(* CODESYS project ElevatorProblem.project

Project tree, tasks and I/O mapping:
  Device : Elmo Platinum Maestro, Elmo Motion Control, version 1.0.0.2
    application Application
      libraries: Standard, * (System)
      task MainTask (cyclic, interval t#100ms, priority 1) calls PLC_PRG, PLC_PRG
      task VISU_TASK (cyclic, interval 100 ms, priority 31) calls VisuElems.Visu_Prg
      program PLC_PRG [ST]
      01_Enumerator/
        data type eFloor
        data type eMOVESTOP
        data type eElevatorType
        data type eButton
        data type eUPDOWN
      02_Structure/
        data type stElevator
        data type stFloor
        data type stFloorRequest
      03_Module/
        function block FB_Elevator [ST]: M_ColorElevator, pCurrentFloor, M_Move, M_ButtonClicked, pColorButtons, pDestinPos, pB1Invisible, M_ShowClickedButton, M_FloorReached, M_DetermineNextFloor, pCurrentRequest, pMoving, pDirection, pCurrentDestin, pRequest, pCurrentPos, pCurrentPeople, pMaxPeople
        function block FB_ElevatorGuests [ST]: pColorButtons, pB1Invisible, pMaxPeople
        function block FB_Floor [ST]: pTopInvisible, pBottomInvisible, pFloorNumber, pPeople
        function block FB_FloorTop [ST]: pTopInvisible
        function block FB_FloorBottom [ST]: pBottomInvisible
        function block FB_Building [ST]: M_RequestExecuted, pFloorRequestedQueue, M_NewFloorRequest, M_AssignElevators, M_Distance
      visualisation Visualization
      visualisation Elevator
      visualisation Floor
    Elmo_Master_Device : Elmo Master Device, Elmo, version 1.0.0.2
  libraries: VisuSymbols, 3.5.10.0 (System)
  text list GlobalTextList
*)

// Device/Application/01_Enumerator/eFloor
TYPE eFloor :
(
	Wait := -1,
	B1 := 0,
	F1 := 1,
	F2 := 2,
	F3 := 3,
	F4 := 4,
	F5 := 5
);
END_TYPE

// Device/Application/01_Enumerator/eMOVESTOP
TYPE eMOVESTOP :
(
	WAITING := 0, // doors are open -> people can get on and off
	MOVING := 1,
	STOPPING := 2
);
END_TYPE

// Device/Application/02_Structure/stElevator
TYPE stElevator :
STRUCT
	uiElevatorType : UINT;
	dwColorElevator : DWORD;
	dwColorButtons : DWORD;
	uiCurrentPos : UINT := 0;
	iDestinPos : UINT := 0;
	uiCurrentPeople : UINT;
	uiCurrentFloor : eFloor;
	xMoving : BOOL;
	xB1Access : BOOL;
	
	// Bools and trigger for buttons
	trig_ButtonF1 : R_Trig;
	xF1 : BOOL;
	xF1Clicked : BOOL;
	trig_ButtonF2 : R_Trig;
	xF2 : BOOL;
	xF2Clicked : BOOL;
	trig_ButtonF3 : R_Trig;
	xF3 : BOOL;
	xF3Clicked : BOOL;
	trig_ButtonF4 : R_Trig;
	xF4 : BOOL;
	xF4Clicked : BOOL;
	trig_ButtonF5 : R_Trig;
	xF5 : BOOL;
	xF5Clicked : BOOL;
	trig_ButtonB1 : R_Trig;
	xB1 : BOOL;
	xB1Clicked : BOOL;
	trig_ButtonClose : R_Trig;
	xClose : BOOL;
	trig_ButtonOpen : R_Trig;
	xOpen : BOOL;
		
END_STRUCT
END_TYPE

// Device/Application/01_Enumerator/eElevatorType
{attribute 'qualified_only'}
{attribute 'strict'}
TYPE eElevatorType :
(
	GUEST := 1,
	FREIGHT := 0
);
END_TYPE

// Device/Application/02_Structure/stFloor
TYPE stFloor :
STRUCT
	uiFloorNumber : UINT;
	uiPeople : UINT;
	
	xTopInvisible : BOOL;
	xBottomInvisible : BOOL;
	
	trig_ButtonUP : R_Trig;
	xUP : BOOL;
	xUpClicked : BOOL;
	trig_ButtonDOWN : R_Trig;
	xDOWN : BOOL;
	xDownClicked : BOOL;
	
	trig_ButtonPeople : R_Trig;
	xPeople : BOOL;
	trig_ButtonPeopleMinus : R_Trig;
	xPeopleMinus : BOOL;
	
END_STRUCT
END_TYPE

// Device/Application/01_Enumerator/eButton
{attribute 'qualified_only'}
{attribute 'strict'}
TYPE eButton :
(
	B1 := 0,
	F1 := 1,
	F2 := 2,
	F3 := 3,
	F4 := 4,
	F5 := 5,
	CLOSE := 6,
	OPEN := 7
);
END_TYPE

// Device/Application/01_Enumerator/eUPDOWN
{attribute 'qualified_only'}
{attribute 'strict'}
TYPE eUPDOWN :
(
	Wait := -1,
	UP := 0,
	DOWN := 1
);
END_TYPE

// Device/Application/02_Structure/stFloorRequest
TYPE stFloorRequest :
STRUCT
	eFloor : eFloor := -1;
    eUPDOWN : eUPDOWN := -1;
END_STRUCT
END_TYPE

// Device/Application/PLC_PRG
PROGRAM PLC_PRG
VAR
	(* Object declarations *)
	fbElevatorGuests : ARRAY [1..uiObject] OF FB_ElevatorGuests; // Elevator 1 and 2
	stElevatorGuestsData : ARRAY [1..uiObject] OF stElevator;	// Data for elevator 1 and 2
	
	fbElevator : FB_Elevator;	// Elevator 3
	stElevatorData : stElevator;	// Data for Elevator 3
	
	fbBuilding : FB_Building;	// Building
	fbAllElevators : ARRAY [1..3] OF FB_Elevator;	// Array with all Elevators of Building
	fbAllFloors : ARRAY[0..5] OF FB_Floor;
	
	fbFloor : ARRAY [1..uiObjectFloor] OF FB_Floor;	// Floors 1 to 4
	stFloorData : ARRAY [1..uiObjectFloor] OF stFLoor;	// Data for Floor 1 to 4
	
	fbFloorTop : FB_FloorTop;	// Floor 5
	stFloorTopData : stFloor;	// Data for Floor 5
	
	fbFloorBottom : FB_FloorBottom;	// Floor B1 aka 0
	stFloorBottomData : stFloor;	// Data for Floor B1
	
	(* Variables for handling elevator movements and requests *)
	xButtonsClicked : ARRAY[0..5] OF BOOL;	// Array for clicked buttons
	CommandToElevator : ARRAY [1..3] OF stFloorRequest;	// Array for Floor Requests to Elevator
	
	// new Floor Requests
	stNewFloorRequest : stFloorRequest;
	eRequestedFloor : stFloorRequest;
	xFloorRequestClicked : ARRAY[1..10] OF BOOL;
	
	// helper variables
	iCnt : UINT;	// counter Variable
	uiPeopleElevators : ARRAY[1..3] OF UINT;
	uiPeopleFloors : ARRAY[0..5] OF UINT;
	

	
END_VAR
VAR CONSTANT
	uiObject : UINT := 2;
	uiObjectFloor : UINT :=4;
END_VAR

// FLOORS
FOR iCnt := 1 TO uiObjectFloor BY 1 DO
	fbFloor[iCnt].pFloorNumber := iCnt;
	stFloorData[iCnt].uiPeople := fbFloor[iCnt].pPeople;
	stFloorData[iCnt].uiFloorNumber := fbFloor[iCnt].pFloorNumber;
	stFloorData[iCnt].xBottomInvisible := fbFloor[iCnt].pBottomInvisible;
	stFloorData[iCnt].xTopInvisible := fbFloor[iCnt].pTopInvisible;
	stFloorData[iCnt].trig_ButtonDOWN(CLK := stFloorData[iCnt].xDOWN);
	stFloorData[iCnt].trig_ButtonUP(CLK := stFloorData[iCnt].xUP);
	stFloorData[iCnt].trig_ButtonPeople(CLK := stFloorData[iCnt].xPeople);
	stFloorData[iCnt].trig_ButtonPeopleMinus(CLK := stFloorData[iCnt].xPeopleMinus);
	IF stFloorData[iCnt].trig_ButtonDOWN.Q THEN
		stNewFloorRequest.eFloor := fbFloor[iCnt].pFloorNumber;
		stNewFloorRequest.eUPDOWN := eUPDOWN.DOWN;
		fbBuilding.M_NewFloorRequest(stNewFloorRequest);
		xFloorRequestClicked[iCnt*2] := TRUE;
	ELSIF stFloorData[iCnt].trig_ButtonUP.Q THEN
		stNewFloorRequest.eFloor := fbFloor[iCnt].pFloorNumber;
		stNewFloorRequest.eUPDOWN := eUPDOWN.UP;
		fbBuilding.M_NewFloorRequest(stNewFloorRequest);
		xFloorRequestClicked[(iCnt*2)+1] := TRUE;
	END_IF
	IF stFloorData[iCnt].trig_ButtonPeople.Q THEN
		fbFloor[iCnt].pPeople := fbFloor[iCnt].pPeople + 1;
	END_IF
	IF stFloorData[iCnt].trig_ButtonPeopleMinus.Q THEN
		IF fbFloor[iCnt].pPeople > 0 THEN
			fbFloor[iCnt].pPeople := fbFloor[iCnt].pPeople - 1;
		END_IF
	END_IF
	stFloorData[iCnt].xDownClicked := xFloorRequestClicked[iCnt*2];
	stFloorData[iCnt].xUpClicked := xFloorRequestClicked[(iCnt*2)+1];
	
	
END_FOR
// Top Floor
fbFloorTop.pFloorNumber := 5;
stFloorTopData.uiPeople := fbFloorTop.pPeople;
stFloorTopData.uiFloorNumber := fbFloorTop.pFloorNumber;
stFloorTopData.xBottomInvisible := fbFloorTop.pBottomInvisible;
stFloorTopData.xTopInvisible := fbFloorTop.pTopInvisible;
stFloorTopData.trig_ButtonDOWN(CLK := stFloorTopData.xDOWN);
stFloorTopData.trig_ButtonPeople(CLK := stFloorTopData.xPeople);
stFloorTopData.trig_ButtonPeopleMinus(CLK := stFloorTopData.xPeopleMinus);
IF stFloorTopData.trig_ButtonDOWN.Q THEN
	stNewFloorRequest.eFloor := fbFloorTop.pFloorNumber;
	stNewFloorRequest.eUPDOWN := eUPDOWN.DOWN;
	fbBuilding.M_NewFloorRequest(stNewFloorRequest);
	xFloorRequestClicked[10] := TRUE;
END_IF
IF stFloorTopData.trig_ButtonPeople.Q THEN
	fbFloorTop.pPeople := fbFloorTop.pPeople + 1;
END_IF
IF stFloorTopData.trig_ButtonPeopleMinus.Q THEN
	IF fbFloorTop.pPeople > 0 THEN
		fbFloorTop.pPeople := fbFloorTop.pPeople - 1;
	END_IF
END_IF
stFloorTopData.xDownClicked := xFloorRequestClicked[10];
// Bottom Floor
fbFloorBottom.pFloorNumber := 0;
stFloorBottomData.uiPeople := fbFloorBottom.pPeople;
stFloorBottomData.uiFloorNumber := fbFloorBottom.pFloorNumber;
stFloorBottomData.xBottomInvisible := fbFloorBottom.pBottomInvisible;
stFloorBottomData.xTopInvisible := fbFloorBottom.pTopInvisible;
stFloorBottomData.trig_ButtonUP(CLK := stFloorBottomData.xUP);
stFloorBottomData.trig_ButtonPeople(CLK := stFloorBottomData.xPeople);
stFloorBottomData.trig_ButtonPeopleMinus(CLK := stFloorBottomData.xPeopleMinus);
IF stFloorBottomData.trig_ButtonUP.Q THEN
	stNewFloorRequest.eFloor := fbFloorBottom.pFloorNumber;
	stNewFloorRequest.eUPDOWN := eUPDOWN.UP;
	fbBuilding.M_NewFloorRequest(stNewFloorRequest);
	xFloorRequestClicked[1] := TRUE;
END_IF
IF stFloorBottomData.trig_ButtonPeople.Q THEN
	fbFloorBottom.pPeople := fbFloorBottom.pPeople + 1;
END_IF
IF stFloorBottomData.trig_ButtonPeopleMinus.Q THEN
	IF fbFloorBottom.pPeople > 0 THEN
		fbFloorBottom.pPeople := fbFloorBottom.pPeople - 1;
	END_IF
END_IF
stFloorBottomData.xUpClicked := xFloorRequestClicked[1];



// Building
fbAllFloors[0] := fbFloorBottom;
fbAllFloors[1] := fbFloor[1];
fbAllFloors[2] := fbFloor[2];
fbAllFloors[3] := fbFloor[3];
fbAllFloors[4] := fbFloor[4];
fbAllFloors[5] := fbFloorTop;
fbBuilding.fbFloors := fbAllFloors;
fbAllElevators[1] := fbElevatorGuests[1];
fbAllElevators[2] := fbElevatorGuests[2];
fbAllElevators[3] := fbElevator;
fbBuilding.fbElevators := fbAllElevators;
CommandToElevator := fbBuilding.M_AssignElevators();

// ELEVATORS
// guest elevators
FOR iCnt := 1 TO uiObject BY 1 DO
	// Floor Request
	fbElevatorGuests[iCnt].pCurrentRequest := CommandToElevator[iCnt];
	IF CommandToElevator[iCnt].eFloor <> -1 THEN
		fbElevatorGuests[iCnt].pRequest := TRUE;
		fbElevatorGuests[iCnt].M_DetermineNextFloor();
		fbAllElevators[1] := fbElevatorGuests[1];
		fbAllElevators[2] := fbElevatorGuests[2];
		fbBuilding.fbElevators := fbAllElevators;
	ELSE
		fbElevatorGuests[iCnt].pRequest := FALSE;
	END_IF

	// transfer of general data from the object to the visualization struct
	stElevatorGuestsData[iCnt].xB1Access := fbElevatorGuests[iCnt].pB1Invisible;
	stElevatorGuestsData[iCnt].uiCurrentFloor := fbElevatorGuests[iCnt].pCurrentFloor;
	stElevatorGuestsData[iCnt].dwColorElevator := fbElevatorGuests[iCnt].M_ColorElevator();
	stElevatorGuestsData[iCnt].dwColorButtons := fbElevatorGuests[iCnt].pColorButtons;
	stElevatorGuestsData[iCnt].uiCurrentPeople := fbElevatorGuests[iCnt].pCurrentPeople;
	// MOVE
	stElevatorGuestsData[iCnt].uiCurrentPos := fbElevatorGuests[iCnt].M_Move();

	// Buttons configuration
	stElevatorGuestsData[iCnt].xMoving := fbElevatorGuests[iCnt].xMoving;
	stElevatorGuestsData[iCnt].trig_ButtonF1(CLK := stElevatorGuestsData[iCnt].xF1);
	stElevatorGuestsData[iCnt].trig_ButtonF2(CLK := stElevatorGuestsData[iCnt].xF2);
	stElevatorGuestsData[iCnt].trig_ButtonF3(CLK := stElevatorGuestsData[iCnt].xF3);
	stElevatorGuestsData[iCnt].trig_ButtonF4(CLK := stElevatorGuestsData[iCnt].xF4);
	stElevatorGuestsData[iCnt].trig_ButtonF5(CLK := stElevatorGuestsData[iCnt].xF5);
	stElevatorGuestsData[iCnt].trig_ButtonB1(CLK := stElevatorGuestsData[iCnt].xB1);
	stElevatorGuestsData[iCnt].trig_ButtonClose(CLK := stElevatorGuestsData[iCnt].xClose);
	stElevatorGuestsData[iCnt].trig_ButtonOpen(CLK := stElevatorGuestsData[iCnt].xOpen);
	IF stElevatorGuestsData[iCnt].trig_ButtonF1.Q THEN
		fbElevatorGuests[iCnt].iiPressedButton := eButton.F1;
		fbElevatorGuests[iCnt].M_ButtonClicked(fbElevatorGuests[iCnt].iiPressedButton);
	ELSIF stElevatorGuestsData[iCnt].trig_ButtonF2.Q THEN
		fbElevatorGuests[iCnt].iiPressedButton := eButton.F2;
		fbElevatorGuests[iCnt].M_ButtonClicked(fbElevatorGuests[iCnt].iiPressedButton);
	ELSIF stElevatorGuestsData[iCnt].trig_ButtonF3.Q THEN
		fbElevatorGuests[iCnt].iiPressedButton := eButton.F3;
		fbElevatorGuests[iCnt].M_ButtonClicked(fbElevatorGuests[iCnt].iiPressedButton);
	ELSIF stElevatorGuestsData[iCnt].trig_ButtonF4.Q THEN
		fbElevatorGuests[iCnt].iiPressedButton := eButton.F4;
		fbElevatorGuests[iCnt].M_ButtonClicked(fbElevatorGuests[iCnt].iiPressedButton);
	ELSIF stElevatorGuestsData[iCnt].trig_ButtonF5.Q THEN
		fbElevatorGuests[iCnt].iiPressedButton := eButton.F5;
		fbElevatorGuests[iCnt].M_ButtonClicked(fbElevatorGuests[iCnt].iiPressedButton);
	ELSIF stElevatorGuestsData[iCnt].trig_ButtonB1.Q THEN
		fbElevatorGuests[iCnt].iiPressedButton := eButton.B1;
		fbElevatorGuests[iCnt].M_ButtonClicked(fbElevatorGuests[iCnt].iiPressedButton);
	ELSIF stElevatorGuestsData[iCnt].trig_ButtonClose.Q THEN
		fbElevatorGuests[iCnt].iiPressedButton := eButton.CLOSE;
		fbElevatorGuests[iCnt].M_ButtonClicked(fbElevatorGuests[iCnt].iiPressedButton);
	ELSIF stElevatorGuestsData[iCnt].trig_ButtonOpen.Q THEN
		fbElevatorGuests[iCnt].iiPressedButton := eButton.OPEN;
		fbElevatorGuests[iCnt].M_ButtonClicked(fbElevatorGuests[iCnt].iiPressedButton);
	ELSE
		fbElevatorGuests[iCnt].iiPressedButton := -1;
	END_IF
	
	// Remove request if executed ( if the current status of Requested is False, but before Move() it was true)
	IF NOT fbElevatorGuests[iCnt].pRequest AND fbAllElevators[iCnt].pRequest THEN
		eRequestedFloor := fbElevatorGuests[iCnt].pCurrentRequest;
		IF fbElevatorGuests[iCnt].pCurrentFloor = eRequestedFloor.eFloor THEN
			fbBuilding.M_RequestExecuted(eRequestedFloor);
			// update people on all floors and elevators
			
			uiPeopleElevators := fbBuilding.PeopleToElevator;
			fbElevatorGuests[1].pCurrentPeople := uiPeopleElevators[1];
			fbElevatorGuests[2].pCurrentPeople := uiPeopleElevators[2];
			fbElevator.pCurrentPeople := uiPeopleElevators[3];
			uiPeopleFloors := fbBuilding.PeopleToFloor;
			fbFloorBottom.pPeople := uiPeopleFloors[0];
			fbFloor[1].pPeople := uiPeopleFloors[1];
			fbFloor[2].pPeople := uiPeopleFloors[2];
			fbFloor[3].pPeople := uiPeopleFloors[3];
			fbFloor[4].pPeople := uiPeopleFloors[4];
			fbFloorTop.pPeople := uiPeopleFloors[5];
			
		END_IF
		// untoggle Floor button (F1-F4)
		IF eRequestedFloor.eFloor > eFloor.B1 AND eRequestedFloor.eFloor < eFloor.F5 THEN
			IF eRequestedFloor.eUPDOWN = eUPDOWN.DOWN THEN
				stFloorData[eRequestedFloor.eFloor].xDOWN := FALSE;
				xFloorRequestClicked[eRequestedFloor.eFloor*2] := FALSE;
			ELSIF eRequestedFloor.eUPDOWN = eUPDOWN.UP THEN
				stFloorData[eRequestedFloor.eFloor].xUP := FALSE;
				xFloorRequestClicked[eRequestedFloor.eFloor*2+1] := FALSE;
			END_IF
			// shouldn't happen because not reachable for guest elevators
		ELSIF eRequestedFloor.eFloor = eFloor.B1 THEN
			stFloorBottomData.xUP := FALSE;
			xFloorRequestClicked[1] := FALSE;
		ELSIF eRequestedFloor.eFloor = eFloor.F5 THEN
			stFloorTopData.xDOWN := FALSE;
			xFloorRequestClicked[10] := FALSE;
		END_IF		
	END_IF
	
	// Button style
	xButtonsClicked := fbElevatorGuests[iCnt].M_ShowClickedButton();
	stElevatorGuestsData[iCnt].xB1Clicked := xButtonsClicked[0];
	stElevatorGuestsData[iCnt].xF1Clicked := xButtonsClicked[1];
	stElevatorGuestsData[iCnt].xF2Clicked := xButtonsClicked[2];
	stElevatorGuestsData[iCnt].xF3Clicked := xButtonsClicked[3];
	stElevatorGuestsData[iCnt].xF4Clicked := xButtonsClicked[4];
	stElevatorGuestsData[iCnt].xF5Clicked := xButtonsClicked[5];
	
END_FOR

//  Freight Elevator 
// Floor request
IF CommandToElevator[3].eFloor <> -1 THEN
	fbElevator.pCurrentRequest := CommandToElevator[3];
	fbElevator.pRequest := TRUE;
	fbElevator.M_DetermineNextFloor();
	fbAllElevators[3] := fbElevator;
	fbBuilding.fbElevators := fbAllElevators;
END_IF
// general properites
stElevatorData.xB1Access := fbElevator.pB1Invisible;
stElevatorData.uiCurrentFloor := fbElevator.pCurrentFloor;
stElevatorData.dwColorElevator := fbElevator.M_ColorElevator();
stElevatorData.dwColorButtons := fbElevator.pColorButtons;
stElevatorData.uiCurrentPeople := fbElevator.pCurrentPeople;
// MOVE
stElevatorData.uiCurrentPos := fbElevator.M_Move();
// Button linking
stElevatorData.xMoving := fbElevator.xMoving;
stElevatorData.trig_ButtonF1(CLK := stElevatorData.xF1);
stElevatorData.trig_ButtonF2(CLK := stElevatorData.xF2);
stElevatorData.trig_ButtonF3(CLK := stElevatorData.xF3);
stElevatorData.trig_ButtonF4(CLK := stElevatorData.xF4);
stElevatorData.trig_ButtonF5(CLK := stElevatorData.xF5);
stElevatorData.trig_ButtonB1(CLK := stElevatorData.xB1);
stElevatorData.trig_ButtonClose(CLK := stElevatorData.xClose);
stElevatorData.trig_ButtonOpen(CLK := stElevatorData.xOpen);
IF stElevatorData.trig_ButtonF1.Q THEN
	fbElevator.iiPressedButton := eButton.F1;
	fbElevator.M_ButtonClicked(fbElevator.iiPressedButton);
ELSIF stElevatorData.trig_ButtonF2.Q THEN
	fbElevator.iiPressedButton := eButton.F2;
	fbElevator.M_ButtonClicked(fbElevator.iiPressedButton);
ELSIF stElevatorData.trig_ButtonF3.Q THEN
	fbElevator.iiPressedButton := eButton.F3;
	fbElevator.M_ButtonClicked(fbElevator.iiPressedButton);
ELSIF stElevatorData.trig_ButtonF4.Q THEN
	fbElevator.iiPressedButton := eButton.F4;
	fbElevator.M_ButtonClicked(fbElevator.iiPressedButton);
ELSIF stElevatorData.trig_ButtonF5.Q THEN
	fbElevator.iiPressedButton := eButton.F5;
	fbElevator.M_ButtonClicked(fbElevator.iiPressedButton);
ELSIF stElevatorData.trig_ButtonB1.Q THEN
	fbElevator.iiPressedButton := eButton.B1;
	fbElevator.M_ButtonClicked(fbElevator.iiPressedButton);
ELSIF stElevatorData.trig_ButtonClose.Q THEN
	fbElevator.iiPressedButton := eButton.CLOSE;
	fbElevator.M_ButtonClicked(fbElevator.iiPressedButton);
ELSIF stElevatorData.trig_ButtonOpen.Q THEN
	fbElevator.iiPressedButton := eButton.OPEN;
	fbElevator.M_ButtonClicked(fbElevator.iiPressedButton);
ELSE
	fbElevator.iiPressedButton := -1;
END_IF
// button style depending on clicked or not
xButtonsClicked := fbElevator.M_ShowClickedButton();
stElevatorData.xB1Clicked := xButtonsClicked[0];
stElevatorData.xF1Clicked := xButtonsClicked[1];
stElevatorData.xF2Clicked := xButtonsClicked[2];
stElevatorData.xF3Clicked := xButtonsClicked[3];
stElevatorData.xF4Clicked := xButtonsClicked[4];
stElevatorData.xF5Clicked := xButtonsClicked[5];

// Remove request if executed
IF NOT fbElevator.pRequest AND fbAllElevators[3].pRequest THEN
	eRequestedFloor := fbElevator.pCurrentRequest;
	IF fbElevator.pCurrentFloor = eRequestedFloor.eFloor THEN
		fbBuilding.M_RequestExecuted(eRequestedFloor);// update people on all floors and elevators
		uiPeopleElevators := fbBuilding.PeopleToElevator;
		fbElevatorGuests[1].pCurrentPeople := uiPeopleElevators[1];
		fbElevatorGuests[2].pCurrentPeople := uiPeopleElevators[2];
		fbElevator.pCurrentPeople := uiPeopleElevators[3];
		uiPeopleFloors := fbBuilding.PeopleToFloor;
		fbFloorBottom.pPeople := uiPeopleFloors[0];
		fbFloor[1].pPeople := uiPeopleFloors[1];
		fbFloor[2].pPeople := uiPeopleFloors[2];
		fbFloor[3].pPeople := uiPeopleFloors[3];
		fbFloor[4].pPeople := uiPeopleFloors[4];
		fbFloorTop.pPeople := uiPeopleFloors[5];
	END_IF
	// untoggle Floor button (F1-F4)
	IF eRequestedFloor.eFloor > eFloor.B1 AND eRequestedFloor.eFloor < eFloor.F5 THEN
		IF eRequestedFloor.eUPDOWN = eUPDOWN.DOWN THEN
			stFloorData[eRequestedFloor.eFloor].xDOWN := FALSE;
			xFloorRequestClicked[eRequestedFloor.eFloor*2] := FALSE;
		ELSIF eRequestedFloor.eUPDOWN = eUPDOWN.UP THEN
			stFloorData[eRequestedFloor.eFloor].xUP := FALSE;
			xFloorRequestClicked[eRequestedFloor.eFloor*2+1] := FALSE;
		END_IF
	ELSIF eRequestedFloor.eFloor = eFloor.B1 THEN
		stFloorBottomData.xUP := FALSE;
		xFloorRequestClicked[1] := FALSE;
	ELSIF eRequestedFloor.eFloor = eFloor.F5 THEN
		stFloorTopData.xDOWN := FALSE;
		xFloorRequestClicked[10] := FALSE;
	END_IF
END_IF

END_PROGRAM

// Device/Application/03_Module/FB_ElevatorGuests
FUNCTION_BLOCK FB_ElevatorGuests EXTENDS FB_Elevator
VAR_INPUT
END_VAR
VAR_OUTPUT
END_VAR
VAR
	
END_VAR

SUPER^();

PROPERTY pColorButtons : DWORD
GET
pColorButtons := 16#FFE227F5; // purple
END_GET
END_PROPERTY

PROPERTY pB1Invisible : BOOL
GET
pB1Invisible := TRUE;
END_GET
END_PROPERTY

PROPERTY pMaxPeople : UINT
GET
pMaxPeople := 3;
END_GET
END_PROPERTY

END_FUNCTION_BLOCK

// Device/Application/03_Module/FB_Elevator
FUNCTION_BLOCK FB_Elevator 
VAR_INPUT
	iiPressedButton : INT;
END_VAR
VAR_OUTPUT
END_VAR
VAR
	xElevatorGuests : BOOL;
	uiCurrentPos : UINT := 0;
	uiDestinPos : UINT := 0;
	
	iWaitCnt : INT := 300;
	
	eNextFloor : eFloor := -1;
	eCurrentFloor : eFloor;
	eMovingDirection : eUPDOWN := eUPDOWN.DOWN;
	uiMoveStop : eMOVESTOP := eMOVESTOP.WAITING;
	xMoving : BOOL;
	
	// clicked Buttons:
	xClickedButtons : ARRAY [0..5] OF BOOL;
	iLoop : INT;  // Loop index
	bFound : BOOL := FALSE;  // Flag to indicate if the next floor is found
	
	// requested Floors
	stCurrentFloorRequest : stFloorRequest;
	xRequested : BOOL := FALSE;
	
	// PEOPLE
	uiCurrentPeople : UINT;
	uiMaxPeople : UINT := 5;
	
END_VAR

METHOD M_ColorElevator : DWORD
VAR_INPUT
END_VAR
CASE uiMoveStop OF
eMOVESTOP.MOVING:
	M_ColorElevator := 16#AA000000;
eMOVESTOP.STOPPING:
	M_ColorElevator := 16#AA000000;
ELSE 
	M_ColorElevator := 16#88888888;
END_CASE
END_METHOD

PROPERTY pCurrentFloor : eFloor
GET
IF eMovingDirection = eUPDOWN.DOWN THEN
	IF uiCurrentPos = 0 THEN
		pCurrentFloor := eFloor.F5;
	ELSIF uiCurrentPos > 0 AND uiCurrentPos <= 150 THEN
		pCurrentFloor := eFloor.F4;
	ELSIF uiCurrentPos > 150 AND uiCurrentPos <= 300 THEN
		pCurrentFloor := eFloor.F3;
	ELSIF uiCurrentPos > 300 AND uiCurrentPos <= 450 THEN
		pCurrentFloor := eFloor.F2;
	ELSIF uiCurrentPos > 450 AND uiCurrentPos <= 600 THEN
		pCurrentFloor := eFloor.F1;
	ELSIF uiCurrentPos > 600 AND uiCurrentPos <= 750 THEN
		pCurrentFloor := eFloor.B1;
	END_IF
ELSE
	IF uiCurrentPos >= 0 AND uiCurrentPos < 150 THEN
		pCurrentFloor := eFloor.F5;
	ELSIF uiCurrentPos >= 150 AND uiCurrentPos < 300 THEN
		pCurrentFloor := eFloor.F4;
	ELSIF uiCurrentPos >= 300 AND uiCurrentPos < 450 THEN
		pCurrentFloor := eFloor.F3;
	ELSIF uiCurrentPos >= 450 AND uiCurrentPos < 600 THEN
		pCurrentFloor := eFloor.F2;
	ELSIF uiCurrentPos >= 600 AND uiCurrentPos < 750 THEN
		pCurrentFloor := eFloor.F1;
	ELSIF uiCurrentPos >= 750 THEN
		pCurrentFloor := eFloor.B1;
	END_IF
END_IF
END_GET
END_PROPERTY

METHOD M_Move : UINT
VAR_INPUT
END_VAR
VAR
	xMoved : BOOL;
END_VAR
xMoved := FALSE;
CASE uiMoveStop OF
eMOVESTOP.MOVING:
	xMoving := TRUE;
	FOR iLoop := 0 TO 5 DO
		IF xClickedButtons[iLoop] THEN
			bFound := TRUE;
			EXIT;
		END_IF
	END_FOR
	IF NOT bFound AND NOT pRequest THEN
		// stop at next floor
		CASE pCurrentFloor OF
		eFLOOR.B1:
			uiDestinPos := 750;
		eFLOOR.F1:
			uiDestinPos := 600;
		eFLOOR.F2:
			uiDestinPos := 450;
		eFLOOR.F3:
			uiDestinPos := 300;
		eFLOOR.F4:
			uiDestinPos := 150;
		eFLOOR.F5:
			uiDestinPos := 0;
		END_CASE
	END_IF
	
	// MOVE
	IF uiCurrentPos > uiDestinPos THEN //higher number of y-coordinate the lower one goes
		uiCurrentPos := uiCurrentPos - 1;
		eMovingDirection := eUPDOWN.UP;
		xMoved := TRUE;
	ELSIF uiCurrentPos < uiDestinPos THEN
		uiCurrentPos := uiCurrentPos + 1;
		eMovingDirection := eUPDOWN.DOWN;
		xMoved := TRUE;
	END_IF
	IF uiCurrentPos = uiDestinPos AND (xMoved OR pRequest) THEN
		(* if no button clicked and no floor requested, change to stopping mode, otherwise change to floor reached*)
		M_FloorReached();
	ELSIF NOT xMoved THEN
		uiMoveStop := eMOVESTOP.STOPPING; 
		xMoving := FALSE;
	END_IF

	
eMOVESTOP.WAITING:
	xMoving := FALSE;
	IF iWaitCnt = 0 THEN
		M_DetermineNextFloor();
		// check if any floor is requested
		FOR iLoop := 0 TO 5 DO
			IF xClickedButtons[iLoop] THEN
				bFound := TRUE;
				EXIT;
			END_IF
    	END_FOR
		IF uiCurrentPos > uiDestinPos OR uiCurrentPos < uiDestinPos OR bFound THEN
			uiMoveStop := eMOVESTOP.MOVING;
		ELSE
			uiMoveStop := eMOVESTOP.STOPPING;	
		END_IF
		iWaitCnt := -1;
	ELSE
		iWaitCnt:= iWaitCnt - 1;
	END_IF

eMOVESTOP.STOPPING:
	xMoving := FALSE;
	// check if any floor is requested
	FOR iLoop := 0 TO 5 DO
		IF xClickedButtons[iLoop] THEN
			bFound := TRUE;
			EXIT;
		END_IF
	END_FOR
	IF bFound OR pRequest THEN
		uiMoveStop := eMOVESTOP.MOVING;
	END_IF
END_CASE 

M_Move := uiCurrentPos;
END_METHOD

METHOD M_ButtonClicked 
VAR_INPUT
	iiPressedButton : INT;
END_VAR
CASE iiPressedButton OF
eButton.B1:
	xClickedButtons[eFloor.B1] := TRUE;
	iWaitCnt := 300;
//	uiMoveStop := eMOVESTOP.WAITING;
eButton.F1:
	xClickedButtons[eFloor.F1] := TRUE;
	iWaitCnt := 300;
//	uiMoveStop := eMOVESTOP.WAITING;
eButton.F2:
	xClickedButtons[eFloor.F2] := TRUE;
	iWaitCnt := 300;
//	uiMoveStop := eMOVESTOP.WAITING;
eButton.F3:
	xClickedButtons[eFloor.F3] := TRUE;
	iWaitCnt := 300;
//	uiMoveStop := eMOVESTOP.WAITING;
eButton.F4:
	xClickedButtons[eFloor.F4] := TRUE;
	iWaitCnt := 300;
//	uiMoveStop := eMOVESTOP.WAITING;
eButton.F5:
	xClickedButtons[eFloor.F5] := TRUE;
	iWaitCnt := 300;
//	uiMoveStop := eMOVESTOP.WAITING;
eButton.CLOSE:
	uiMoveStop := eMOVESTOP.MOVING;
	iWaitCnt := 20;
eButton.OPEN:
	iWaitCnt := 600;
	uiMoveStop := eMOVESTOP.WAITING;
END_CASE
M_DetermineNextFloor();
M_Move();
END_METHOD

PROPERTY pColorButtons : DWORD
GET
pColorButtons := 16#FFF5AE27;
END_GET
END_PROPERTY

PROPERTY pDestinPos : UINT
SET
uiDestinPos := pDestinPos;
END_SET
GET
pDestinPos := uiDestinPos;
END_GET
END_PROPERTY

PROPERTY pB1Invisible : BOOL
GET
pB1Invisible := FALSE;
END_GET
END_PROPERTY

METHOD M_ShowClickedButton : ARRAY [1..6] OF BOOL
VAR_INPUT
END_VAR
VAR 
	uiFloorPos : UINT;
END_VAR
//
CASE pCurrentFloor OF
eFLOOR.F1:
	IF uiCurrentPos = 600 THEN
		xClickedButtons[1] := FALSE;
	END_IF
eFLOOR.F2:
	IF uiCurrentPos = 450 THEN
		xClickedButtons[2] := FALSE;
	END_IF
eFLOOR.F3:
	IF uiCurrentPos = 300 THEN
		xClickedButtons[3] := FALSE;
	END_IF
eFLOOR.F4:
	IF uiCurrentPos = 150 THEN
		xClickedButtons[4] := FALSE;
	END_IF
eFLOOR.F5:
	IF uiCurrentPos = 0 THEN
		xClickedButtons[5] := FALSE;
	END_IF
eFLOOR.B1:
	IF uiCurrentPos = 750 THEN
		xClickedButtons[0] := FALSE;
	END_IF
END_CASE

M_ShowClickedButton := xClickedButtons;
END_METHOD

METHOD M_FloorReached
VAR_INPUT
END_VAR
IF pCurrentFloor = eNextFloor THEN
	iWaitCnt := 300;
	uiMoveStop := eMOVESTOP.WAITING;
	xMoving := FALSE;
	CASE pCurrentFloor OF
	eFLOOR.F1:
		xClickedButtons[eFloor.F1] := FALSE;
		uiCurrentPeople := 0;
	eFLOOR.F2:
		xClickedButtons[eFloor.F2] := FALSE;
		uiCurrentPeople := 0;
	eFLOOR.F3:
		xClickedButtons[eFloor.F3] := FALSE;
		uiCurrentPeople := 0;
	eFLOOR.F4:
		xClickedButtons[eFloor.F4] := FALSE;
		uiCurrentPeople := 0;
	eFLOOR.F5:
		xClickedButtons[eFloor.F5] := FALSE;
		uiCurrentPeople := 0;
	eFLOOR.B1:
		xClickedButtons[eFloor.B1] := FALSE;
		uiCurrentPeople := 0;
	END_CASE
	IF eNextFloor = stCurrentFloorRequest.eFloor THEN
		pRequest := FALSE;
	END_IF
END_IF
M_DetermineNextFloor();
END_METHOD

METHOD M_DetermineNextFloor
VAR_INPUT
END_VAR
VAR
	xFound : BOOL;
	iDistance : INT;
	eClosestFloor: eFloor;
    iMinDistance: INT;
	
END_VAR
// Initialize the requested floor with the current floor as a default value
eNextFloor := pCurrentFloor;

bFound := FALSE;
CASE eMovingDirection OF
eUPDOWN.UP:
	FOR iLoop := pCurrentFloor TO 5 DO
		IF xClickedButtons[iLoop] THEN
			eNextFloor := iLoop;
			bFound := TRUE;
			EXIT;
		END_IF
	END_FOR
	// If no floor above was found, check for floors below the current floor
	IF NOT bFound THEN
		FOR iLoop := pCurrentFloor - 1 TO 0 BY -1 DO
			IF xClickedButtons[iLoop] THEN
				eNextFloor := iLoop;
				bFound := TRUE;
				EXIT;
			END_IF
		END_FOR
	END_IF

eUPDOWN.DOWN:
	FOR iLoop := pCurrentFloor TO 0 BY -1 DO
		IF xClickedButtons[iLoop] THEN
			eNextFloor := iLoop;
			bFound := TRUE;
			EXIT;
		END_IF
	END_FOR
	// If no floor above was found, check for floors below the current floor
	IF NOT bFound THEN
		FOR iLoop := pCurrentFloor + 1 TO 5 DO
			IF xClickedButtons[iLoop] THEN
				eNextFloor := iLoop;
				bFound := TRUE;
				EXIT;
			END_IF
		END_FOR
	END_IF
END_CASE


IF xRequested THEN
	eNextFloor := stCurrentFloorRequest.eFloor;
(*ELSE
	stCurrentFloorRequest.eFloor := -1;
	stCurrentFloorRequest.eUPDOWN := -1;*)
END_IF

IF (bFound AND iWaitCnt = 0) OR xRequested THEN
	uiMoveStop := eMOVESTOP.MOVING;
END_IF

CASE eNextFloor OF
eFLOOR.B1:
	uiDestinPos := 750;
eFLOOR.F1:
	uiDestinPos := 600;
eFLOOR.F2:
	uiDestinPos := 450;
eFLOOR.F3:
	uiDestinPos := 300;
eFLOOR.F4:
	uiDestinPos := 150;
eFLOOR.F5:
	uiDestinPos := 0;
END_CASE

IF uiDestinPos > uiCurrentPos THEN
	eMovingDirection := eUPDOWN.DOWN;
ELSIF uiDestinPos < uiCurrentPos THEN
	eMovingDirection := eUPDOWN.UP;
END_IF
END_METHOD

PROPERTY pCurrentRequest : stFloorRequest
SET
stCurrentFloorRequest := pCurrentRequest;
END_SET
GET
pCurrentRequest := stCurrentFloorRequest;
END_GET
END_PROPERTY

PROPERTY pMoving : eMOVESTOP
SET
uiMoveStop := pMoving;
END_SET
GET
pMoving := uiMoveStop;
END_GET
END_PROPERTY

PROPERTY pDirection : eUPDOWN
SET
eMovingDirection := pDirection;
END_SET
GET
pDirection := eMovingDirection;
END_GET
END_PROPERTY

PROPERTY pCurrentDestin : eFloor
SET
eNextFloor := pCurrentDestin;
END_SET
GET
pCurrentDestin := eNextFloor;
END_GET
END_PROPERTY

PROPERTY pRequest : BOOL
SET
xRequested := pRequest;
END_SET
GET
pRequest := xRequested;
END_GET
END_PROPERTY

PROPERTY pCurrentPos : UINT
GET
pCurrentPos := uiCurrentPos;
END_GET
END_PROPERTY

PROPERTY pCurrentPeople : UINT
SET
uiCurrentPeople := pCurrentPeople;
END_SET
GET
pCurrentPeople := uiCurrentPeople;
END_GET
END_PROPERTY

PROPERTY pMaxPeople : UINT
GET
pMaxPeople := 5;
END_GET
END_PROPERTY

END_FUNCTION_BLOCK

// Device/Application/03_Module/FB_Building
FUNCTION_BLOCK FB_Building 
VAR_INPUT
	(* Inputs: Requests from each floor and status of elevators *)
//    RequestUp: ARRAY [0..4] OF BOOL; (* Up requests from floors B1 to 4 *)
//    RequestDown: ARRAY [1..5] OF BOOL; (* Down requests from floors 1 to 5 *)
//	sNewFloorRequest : stFloorRequest;
    fbElevators: ARRAY [1..3] OF FB_Elevator; (* Array of elevators *)
	fbFloors : ARRAY [0..5] OF FB_Floor;
END_VAR
VAR_OUTPUT
	(* Outputs: Commands to each elevator *)
    CommandToElevator: ARRAY [1..3] OF stFloorRequest; (* Command to move to a specific floor *)
	PeopleToFloor : ARRAY [0..5] OF UINT;
	PeopleToElevator : ARRAY [1..3] OF UINT;
END_VAR
VAR
	FloorRequestQueue: ARRAY [1..10] OF stFloorRequest; (* Queue of floor requests *)
    QueueStart: INT := 1;
    QueueEnd: INT := 0;
	
	(* Temporary Variables*)
	i: INT;
    AssignedElevator: INT;
    Request: INT;
END_VAR

METHOD M_RequestExecuted
VAR_INPUT
	stExecutedFloor : stFloorRequest;
END_VAR
VAR
    iCnt : INT;
	iElevCnt : INT;
	iShiftCnt : INT;
	stEmptyFloor : stFloorRequest;
	iPplCnt : UINT;
	iPplCnt2 : UINT;
	fbElevator : FB_Elevator;
	stElevatorCurrentRequest : stFloorRequest;
	fbFloor : FB_Floor;
	uiDestinPos : UINT;
	xArrived : BOOL;
	uiMaxPeople : UINT;
END_VAR
PeopleToFloor[0] := fbFloors[0].pPeople;
PeopleToFloor[1] := fbFloors[1].pPeople;
PeopleToFloor[2] := fbFloors[2].pPeople;
PeopleToFloor[3] := fbFloors[3].pPeople;
PeopleToFloor[4] := fbFloors[4].pPeople;
PeopleToFloor[5] := fbFloors[5].pPeople;

FOR iCnt := 1 TO 10 DO
    IF (FloorRequestQueue[iCnt].eFloor = stExecutedFloor.eFloor) AND 
       (FloorRequestQueue[iCnt].eUPDOWN = stExecutedFloor.eUPDOWN) THEN
	   // Assign people to Elevator until Elevaotr full
		// find the Elevator that is on the current Floor
		fbFloor := fbFloors[stExecutedFloor.eFloor];
		CASE stExecutedFloor.eFloor OF 
			eFloor.B1:
				uiDestinPos := 750;
			eFloor.F1:
				uiDestinPos := 600;
			eFloor.F2:
				uiDestinPos := 450;
			eFloor.F3:
				uiDestinPos := 300;
			eFloor.F4:
				uiDestinPos := 150;
			eFloor.F5:
				uiDestinPos := 0;
		END_CASE
		FOR iElevCnt := 1 TO 3 DO
			fbElevator := fbElevators[iElevCnt];
			PeopleToElevator[iElevCnt] := fbElevator.pCurrentPeople;
			stElevatorCurrentRequest := fbElevator.pCurrentRequest;
			xArrived := FALSE;
			IF ((fbElevator.uiCurrentPos <= uiDestinPos AND (uiDestinPos - fbElevator.uiCurrentPos) < 2) OR(fbElevator.uiCurrentPos > uiDestinPos AND (fbElevator.uiCurrentPos - uiDestinPos) < 2)) THEN
				xArrived := TRUE;
			END_IF
			IF stElevatorCurrentRequest.eFloor = stExecutedFloor.eFloor AND stElevatorCurrentRequest.eUPDOWN = stExecutedFloor.eUPDOWN AND xArrived THEN
				iPplCnt2 := 0;
				IF iElevCnt = 3 THEN
					uiMaxPeople := 5;
				ELSE
					uiMaxPeople := 3;
				END_IF
				FOR iPplCnt := 1 TO fbFloor.pPeople DO
					IF PeopleToElevator[iElevCnt] < uiMaxPeople THEN
						PeopleToElevator[iElevCnt] := PeopleToElevator[iElevCnt] + 1;
						iPplCnt2 := iPplCnt2 + 1;
					END_IF
				END_FOR
				PeopleToFloor[stExecutedFloor.eFloor] := PeopleToFloor[stExecutedFloor.eFloor] - iPplCnt2;
			END_IF
		END_FOR
	   
	   	// Request found, shift elements
        FOR iShiftCnt := iCnt TO 9 DO
            FloorRequestQueue[iShiftCnt] := FloorRequestQueue[iShiftCnt + 1];
        END_FOR
		stEmptyFloor.eFloor := eFloor.Wait;
		stEmptyFloor.eUPDOWN := eUPDOWN.Wait;
		FloorRequestQueue[10] := stEmptyFloor;
		QueueEnd := QueueEnd -1;
        RETURN;
    END_IF
END_FOR
END_METHOD

PROPERTY pFloorRequestedQueue : ARRAY [1..10] OF stFloorRequest
SET
END_SET
GET
pFloorRequestedQueue := FloorRequestQueue;
END_GET
END_PROPERTY

METHOD M_NewFloorRequest
VAR_INPUT
	stNewFloorRequest : stFloorRequest;
END_VAR
VAR
	iCnt : UINT;
	iShiftCnt : UINT;
	xExists : BOOL;
	stEmptyFloor : stFloorRequest;
END_VAR
xExists := FALSE;
FOR iCnt := 1 TO QueueEnd DO
	IF stNewFloorRequest.eFloor = FloorRequestQueue[iCnt].eFloor AND stNewFloorRequest.eUPDOWN = FloorRequestQueue[iCnt].eUPDOWN THEN
		xExists := TRUE;
		FOR iShiftCnt := iCnt TO QueueEnd DO
            FloorRequestQueue[iShiftCnt] := FloorRequestQueue[iShiftCnt + 1];
        END_FOR
		stEmptyFloor.eFloor := eFloor.Wait;
		stEmptyFloor.eUPDOWN := eUPDOWN.Wait;
		FloorRequestQueue[10] := stEmptyFloor;
		QueueEnd := QueueEnd -1;
	END_IF
END_FOR

IF NOT xExists THEN
    QueueEnd := QueueEnd + 1;
    FloorRequestQueue[QueueEnd] := stNewFloorRequest;
END_IF
END_METHOD

METHOD M_AssignElevators : ARRAY[1..3] OF stFloorRequest
VAR_INPUT
END_VAR
VAR
	
	stCurrentRequest : stFloorRequest;
	fbCurrentElevator : FB_Elevator;
	iBestElevator : INT; 
	// Helper values
	stTempRequest : stFloorRequest;
	stEmptyRequest : stFloorRequest;
	iFloorCnt: INT;
	iElevatorCnt: INT;
	uiMinDistance : UINT;
	uiDistance : UINT;
	// Flags
	xAssignedElevators : ARRAY[1..3] OF BOOL;
	xCompatibleDirAndPos : BOOL;
END_VAR
// Resetting Arrays
xAssignedElevators[1] := FALSE;
xAssignedElevators[2] := FALSE;
xAssignedElevators[3] := FALSE;
stEmptyRequest.eFloor := -1;
stEmptyRequest.eUPDOWN := -1;
CommandToElevator[1] := stEmptyRequest;
CommandToElevator[2] := stEmptyRequest;
CommandToElevator[3] := stEmptyRequest;


FOR iFloorCnt := 1 TO QueueEnd DO
	// reset all the flags
	stCurrentRequest := FloorRequestQueue[iFloorCnt];
	IF stCurrentRequest.eFloor = -1 THEN
		RETURN;
	END_IF
	iBestElevator := -1;
	uiMinDistance := 999;
	xCompatibleDirAndPos := FALSE;
	// if all elevators are assigned leave loop
	IF xAssignedElevators[1] AND xAssignedElevators[2] AND xAssignedElevators[3] THEN
		RETURN;
	END_IF
	
	FOR iElevatorCnt:= 1 TO 3 DO
		xCompatibleDirAndPos := FALSE;
		// Only iterate elevators that don't have assignment yet
		fbCurrentElevator := fbElevators[iElevatorCnt];
		IF (iElevatorCnt <> 3 AND fbCurrentElevator.pCurrentPeople = 3) OR (iElevatorCnt = 3 AND fbCurrentElevator.pCurrentPeople = 5) THEN
			xAssignedElevators[iElevatorCnt] := TRUE;
		END_IF
		IF xAssignedElevators[iElevatorCnt] = FALSE THEN
			fbCurrentElevator := fbElevators[iElevatorCnt];
			// if B1 Floor then only Elevator 3 
			
			IF stCurrentRequest.eFloor = eFloor.B1 AND iElevatorCnt <> 3 THEN
				iElevatorCnt := 3;
				fbCurrentElevator := fbElevators[iElevatorCnt];
				stTempRequest := fbCurrentElevator.pCurrentRequest;
			END_IF
			// get current distance 
			uiDistance := M_Distance(stCurrentRequest.eFloor, fbCurrentElevator.pCurrentPos);
			// check if elevator is moving BUT only if there is an internal floor request
			IF fbCurrentElevator.pMoving = eMOVESTOP.MOVING THEN
				// check if moving in same direction and floor is on the way to or the current destination IF there is no internal request! 
				stTempRequest := fbCurrentElevator.pCurrentRequest;
				// check if same moving direction
				IF fbCurrentElevator.pDirection = stCurrentRequest.eUPDOWN OR 
					(stTempRequest.eFloor = stCurrentRequest.eFloor AND stTempRequest.eUPDOWN = stCurrentRequest.eUPDOWN) THEN
					// check if on the way to next Floor:
					// Down and between currentPos and destinPos
					IF fbCurrentElevator.pDirection = eUPDOWN.DOWN AND stCurrentRequest.eFloor < fbCurrentElevator.pCurrentFloor AND stCurrentRequest.eFloor > fbCurrentElevator.pCurrentDestin THEN
						xCompatibleDirAndPos := TRUE;
					// Up and between currentPos and destinPos
					ELSIF fbCurrentElevator.pDirection = eUPDOWN.UP AND stCurrentRequest.eFloor > fbCurrentElevator.pCurrentFloor AND stCurrentRequest.eFloor < fbCurrentElevator.pCurrentDestin THEN
						xCompatibleDirAndPos := TRUE;
					// same as destinPos
					ELSIF stCurrentRequest.eFloor = fbCurrentElevator.pCurrentDestin THEN
						xCompatibleDirAndPos := TRUE;
					END_IF
				END_IF
				// if suitible position is found and distance is smaller than previous distance
				IF xCompatibleDirAndPos AND uiDistance < uiMinDistance THEN
					iBestElevator := iElevatorCnt;
					uiMinDistance := uiDistance;
				END_IF
			// if waiting
			ELSIF fbCurrentElevator.pMoving = eMOVESTOP.WAITING THEN
					// Same as currentPos
					IF stCurrentRequest.eFloor = fbCurrentElevator.pCurrentDestin THEN
						xCompatibleDirAndPos := TRUE;
					END_IF
					// if suitible position is found and distance is smaller than previous distance
					IF xCompatibleDirAndPos AND uiDistance < uiMinDistance THEN
						iBestElevator := iElevatorCnt;
						uiMinDistance := uiDistance;
					END_IF
			ELSE // Elevator is not moving
				IF uiDistance < uiMinDistance THEN
					iBestElevator := iElevatorCnt;
					uiMinDistance := uiDistance;
				END_IF
			END_IF		
		END_IF
					
	END_FOR
	IF iBestElevator <> -1 THEN
		CommandToElevator[iBestElevator] := stCurrentRequest;
		xAssignedElevators[iBestElevator] := TRUE;
	END_IF
END_FOR
M_AssignElevators := CommandToElevator;
END_METHOD

METHOD M_Distance : UINT
VAR_INPUT
	ieFloor1 : eFloor;
	iuiPos2 : INT;
END_VAR
VAR
	uiPos1 : INT;
END_VAR
CASE ieFloor1 OF 
	eFloor.B1:
		uiPos1 := 750;
	eFloor.F1:
		uiPos1 := 600;
	eFloor.F2:
		uiPos1 := 450;
	eFloor.F3:
		uiPos1 := 300;
	eFloor.F4:
		uiPos1 := 150;
	eFloor.F5:
		uiPos1 := 0;
END_CASE
M_Distance := ABS(iuiPos2 - uiPos1);
END_METHOD

END_FUNCTION_BLOCK

// Device/Application/03_Module/FB_Floor
FUNCTION_BLOCK FB_Floor
VAR_INPUT
	 ieUpDown : eUPDOWN;
END_VAR
VAR_OUTPUT
END_VAR
VAR
	uiFloorNumber : UINT;
	uiPeople : UINT := 0;
	
	xUP : BOOL;
	xUpClicked : BOOL;
	xDOWN : BOOL;
	XDownClicked : BOOL;
END_VAR

PROPERTY pTopInvisible : BOOL
GET
pTopInvisible := FALSE;
END_GET
END_PROPERTY

PROPERTY pBottomInvisible : BOOL
GET
pBottomInvisible := FALSE;
END_GET
END_PROPERTY

PROPERTY pFloorNumber : UINT
SET
uiFloorNumber := pFloorNumber;
END_SET
GET
pFloorNumber := uiFloorNumber;
END_GET
END_PROPERTY

PROPERTY pPeople : UINT
SET
uiPeople := pPeople;
END_SET
GET
pPeople := uiPeople;
END_GET
END_PROPERTY

END_FUNCTION_BLOCK

// Device/Application/03_Module/FB_FloorTop
FUNCTION_BLOCK FB_FloorTop EXTENDS FB_Floor
VAR_INPUT
END_VAR
VAR_OUTPUT
END_VAR
VAR
END_VAR

SUPER^();

PROPERTY pTopInvisible : BOOL
GET
pTopInvisible := TRUE;
END_GET
END_PROPERTY

END_FUNCTION_BLOCK

// Device/Application/03_Module/FB_FloorBottom
FUNCTION_BLOCK FB_FloorBottom EXTENDS FB_Floor
VAR_INPUT
END_VAR
VAR_OUTPUT
END_VAR
VAR
END_VAR

SUPER^();

PROPERTY pBottomInvisible : BOOL
GET
pBottomInvisible := TRUE;
END_GET
END_PROPERTY

END_FUNCTION_BLOCK

// Device/Application/Visualization
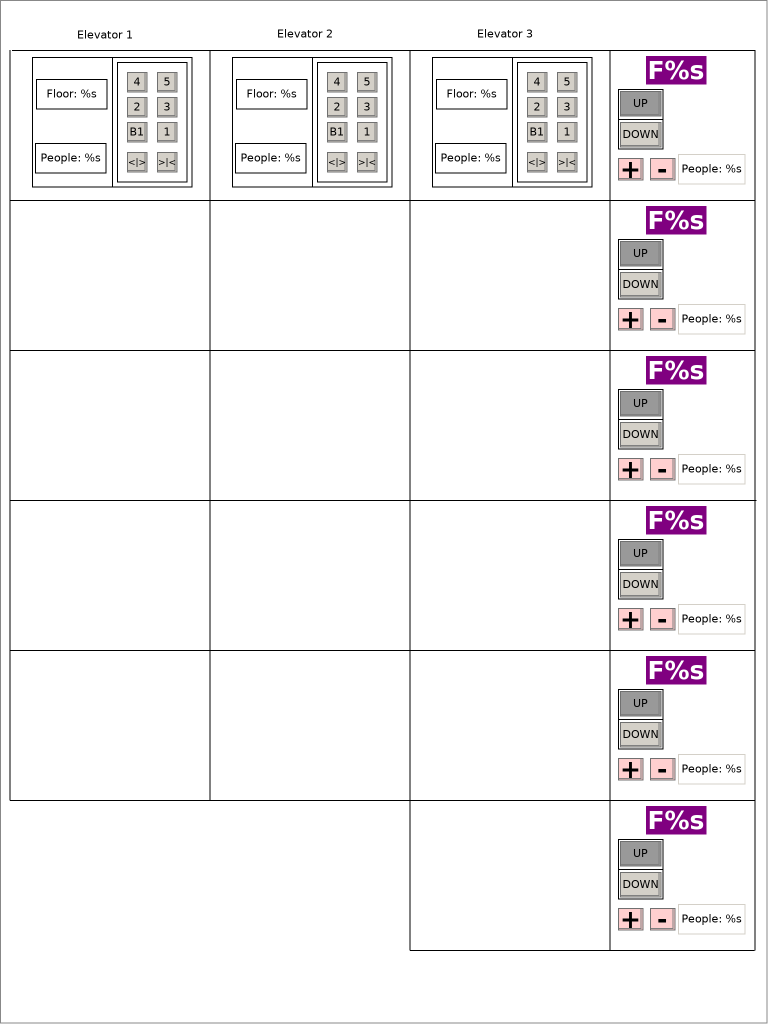
VISUALIZATION Visualization  // 768x1024
    Line (10,800) (10,50)
    Line (210,800) (210,50)
    Line (410,950) (410,50)
    Line (610,950) (610,50)
    Line (610,200) (755,200)
    Line (610,350) (755,350)
    Line (610,800) (755,800)
    Line (10,800) (410,800)
    Line (610,650) (755,650)
    Line (610,500) (756,500)
    Line (410,950) (754,950)
    Line (12,50) (754,50)
    Line (755,950) (755,50)
    Label (30,20 150x30), "Elevator 1"
    Label (230,19 150x30), "Elevator 2"
    Label (430,19 150x30), "Elevator 3"
    Frame (430,55 164x134)
        shows Elevator(stElevatorVisu := PLC_PRG.stElevatorData)
        p2738717112: PLC_PRG.stElevatorData.uiCurrentPos
    Line (10,200) (610,200)
    Line (10,350) (610,350)
    Line (10,500) (610,500)
    Line (10,650) (610,650)
    Line (410,800) (610,800)
    Frame (230,55 164x134)
        shows Elevator(stElevatorVisu := PLC_PRG.stElevatorGuestsData[2])
        p2738717112: PLC_PRG.stElevatorGuestsData[2].uiCurrentPos
    Frame (30,55 164x134)
        shows Elevator(stElevatorVisu := PLC_PRG.stElevatorGuestsData[1])
        p2738717112: PLC_PRG.stElevatorGuestsData[1].uiCurrentPos
    Frame (615,55 134x134)
        shows Floor(stFloorVisu := PLC_PRG.stFloorTopData)
    Frame (615,205 134x134)
        shows Floor(stFloorVisu := PLC_PRG.stFloorData[4])
    Frame (615,355 134x134)
        shows Floor(stFloorVisu := PLC_PRG.stFloorData[3])
    Frame (615,505 134x134)
        shows Floor(stFloorVisu := PLC_PRG.stFloorData[2])
    Frame (615,655 134x134)
        shows Floor(stFloorVisu := PLC_PRG.stFloorData[1])
    Frame (615,805 134x134)
        shows Floor(stFloorVisu := PLC_PRG.stFloorBottomData)
END_VISUALIZATION

// Device/Application/Elevator
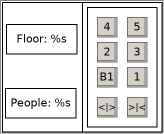
VISUALIZATION Elevator  // 164x134
VAR_IN_OUT
	stElevatorVisu : stElevator;
END_VAR
    Rectangle (2,2 160x130), colour variable: stElevatorVisu.dwColorElevator
    Line (82,2) (82,132)
    RoundedRectangle (6,24 71x30), "Floor: %s", text variable: stElevatorVisu.uiCurrentFloor
    RoundedRectangle (87,7 70x120), colour variable: stElevatorVisu.dwColorButtons
    Button (127,67 20x20), "1", colour toggle: stElevatorVisu.xF1Clicked
        tap stElevatorVisu.xF1
    Button (97,42 20x20), "2", colour toggle: stElevatorVisu.xF2Clicked
        tap stElevatorVisu.xF2
    Button (127,42 20x20), "3", colour toggle: stElevatorVisu.xF3Clicked
        tap stElevatorVisu.xF3
    Button (97,17 20x20), "4", colour toggle: stElevatorVisu.xF4Clicked
        tap stElevatorVisu.xF4
    Button (127,17 20x20), "5", colour toggle: stElevatorVisu.xF5Clicked
        tap stElevatorVisu.xF5
    Button (97,67 20x20), "B1", colour toggle: stElevatorVisu.xB1Clicked, invisible if: stElevatorVisu.xB1Access
        tap stElevatorVisu.xB1
    Button (97,97 20x20), "<|>", input disabled if: stElevatorVisu.xMoving
        tap stElevatorVisu.xOpen
    Button (127,97 20x20), ">|<", input disabled if: stElevatorVisu.xMoving
        tap stElevatorVisu.xClose
    RoundedRectangle (5,88 71x30), "People: %s", text variable: stElevatorVisu.uiCurrentPeople
END_VISUALIZATION

// Device/Application/Floor
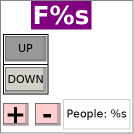
VISUALIZATION Floor  // 134x134
VAR_IN_OUT
	stFloorVisu : stFloor;
END_VAR
    RoundedRectangle (3,34 45x60)
    Line (3,64) (48,64)
    Button (5,36 41x25), "UP", colour toggle: stFloorVisu.xUpClicked, invisible if: stFloorVisu.xTopInvisible
        tap stFloorVisu.xUP
    Button (5,67 41x25), "DOWN", colour toggle: stFloorVisu.xDownClicked, invisible if: stFloorVisu.xBottomInvisible
        tap stFloorVisu.xDOWN
    Textfield (30,0 62x30), "F%s", text variable: stFloorVisu.uiFloorNumber
    Textfield (63,99 67x30), "People: %s", text variable: stFloorVisu.uiPeople
    Button (3,103 25x22), "+"
        tap stFloorVisu.xPeople
    Button (35,103 25x22), "-"
        tap stFloorVisu.xPeopleMinus
END_VISUALIZATION
